SUBAPPLICATION OneSensTwoStateCtrl (* Subapplication Type *)
  (* Standard: 61499-2 *)
  (* Version 1.0, 2020-07-27, AK120569 *)
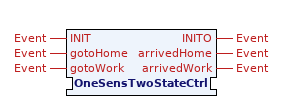
  EVENT_INPUT
    INIT;
    gotoHome;
    gotoWork;
  END_EVENT
  EVENT_OUTPUT
    INITO;
    arrivedHome;
    arrivedWork;
  END_EVENT
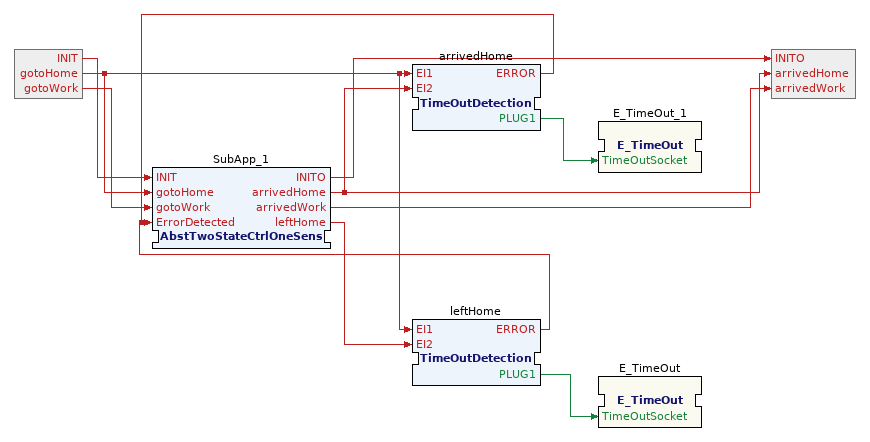
  FBS
    E_TimeOut : E_TimeOut;
    E_TimeOut_1 : E_TimeOut;
  END_FBS
  SUBAPPS
    SubApp_1 : AbstTwoStateCtrlOneSens;
    arrivedHome : TimeOutDetection;
    leftHome : TimeOutDetection;
  END_SUBAPPS
  EVENT_CONNECTIONS
    INIT TO SubApp_1.INIT;
    gotoHome TO SubApp_1.gotoHome;
    gotoWork TO SubApp_1.gotoWork;
    SubApp_1.INITO TO INITO;
    SubApp_1.arrivedHome TO arrivedHome;
    SubApp_1.arrivedWork TO arrivedWork;
    gotoHome TO arrivedHome.EI1;
    SubApp_1.arrivedHome TO arrivedHome.EI2;
    arrivedHome.ERROR TO SubApp_1.ErrorDetected;
    gotoHome TO leftHome.EI1;
    SubApp_1.leftHome TO leftHome.EI2;
    leftHome.ERROR TO SubApp_1.ErrorDetected;
  END_CONNECTIONS
  ADAPTER_CONNECTIONS
    arrivedHome.PLUG1 TO E_TimeOut_1.TimeOutSocket;
    leftHome.PLUG1 TO E_TimeOut.TimeOutSocket;
  END_CONNECTIONS
END_SUBAPPLICATION
